// TIA Portal V20 export
TYPE "SystemSSR"
// stored: Access Published, Namespace LineD1
   STRUCT
      StartSystem : Bool;   // Start the system
      StopSystem : Bool;   // Stop the system
      ResetSystem : Bool;   // Reset the system
   END_STRUCT;
END_TYPE
